{attribute 'qualified_only'}
{attribute 'strict'}
TYPE E_NOTT_CRYO_HEATER_CTRL :
(
	NONE := 0,
	DET_IF, 
	COLD_PLATE,
	PREAMP
);
END_TYPE

(* stored: Version 1.1.0.1, ProductVersion 3.1.4026.18
   DUT E_NOTT_CRYO_HEATER_CTRL: Id {a871dc81-40d0-4f0f-b2d3-ddf496b9c7b5} *)
